(* PLC project Robin example project, CODESYS CODESYS V3.5 SP15, author pdcribeiro *)
(* stored: creationDateTime 2019-12-10T13:33:36.6110185, version 0.0.1, modificationDateTime 2019-12-10T13:33:14.179202, organization INESC TEC *)
(* An example project for the Robin library.

https://github.com/ScalABLE40/robin *)

TYPE TestStruct : STRUCT
  var_bool : BOOL;
  var_byte : BYTE;
  var_int16 : INT;
  var_uint64 : ULINT;
  var_float32 : REAL;
  var_float64 : LREAL;
  var_string : STRING;
  var_pose : Pose;
  var_struct_array : ARRAY[1..10] OF ByteMultiArray;
  {attribute 'robin_var_len'}
  var_struct_varlen_array : ARRAY[1..10] OF ByteMultiArray;
END_STRUCT;
END_TYPE

PROGRAM ROS_PRG
  VAR_INPUT
    double_to_ros : LREAL;
  END_VAR
  VAR_OUTPUT
    double_to_codesys : LREAL;
  END_VAR
  VAR
    robin : Robin;
  END_VAR

                    robin();
// read
robin.read('double_to_codesys', double_to_codesys);
// robin.read('string_varlen_array_to_codesys', string_varlen_array_to_codesys);
// robin.read('struct1_to_codesys', struct1_to_codesys);
// robin.read('struct2_to_codesys', struct2_to_codesys);
// write
robin.write('double_to_ros', double_to_ros);
// robin.write('string_varlen_array_to_ros', string_varlen_array_to_ros);
// robin.write('struct1_to_ros', struct1_to_ros);
// robin.write('struct2_to_ros', struct2_to_ros);

                  
END_PROGRAM

PROGRAM MAIN

                    ROS_PRG.double_to_ros := ROS_PRG.double_to_codesys;
// ROS_PRG.string_varlen_array_to_ros := ROS_PRG.string_varlen_array_to_codesys;
// ROS_PRG.struct1_to_ros := ROS_PRG.struct1_to_codesys;
// ROS_PRG.struct2_to_ros := ROS_PRG.struct2_to_codesys;

                  
END_PROGRAM

CONFIGURATION Device
  RESOURCE Application ON PLC
    TASK MainTask(INTERVAL := T#10ms, PRIORITY := 1);
    PROGRAM MAIN WITH MainTask : MAIN;
    PROGRAM ROS_PRG WITH MainTask : ROS_PRG;
  END_RESOURCE
END_CONFIGURATION

CONFIGURATION SoftMotion General Axis Pool
END_CONFIGURATION
